Staubli VAL3: yes.pgx

public program yes(string x_sMessage (dimensions=1), string& x_sYesNo[] (dimensions=1))
  local num i
  local string l_sButton
begin
  //
  // write a yes no question dialog
  //
  cls()
  if x_sYesNo!=""
    l_sButton[0]=x_sYesNo
  else
    l_sButton[0]="Yes"
  endIf
  // question Dialog
  call questionDialog(x_sMessage,l_sButton,i)
  cls()
  // press F8->YES or ENTER
  //  if i==1 or i==0
  //    x_bResult=true
  //  endIf
end
